        UF : 6, UT : 5,     CONFIG: 'N U T, 0, 0, 0',
       X = -330.7 mm, Y = 229.2 mm, Z = 498.2 mm,
       W = -5.3 deg, P = 20.5 deg,
    GP2:
        UF : 1, UT : 2,
       J1 = 0.0 deg, J2 = 0.0 deg
 };
P[405] {
    GP1:
        UF : 6, UT : 5,     CONFIG: 'N U T, 0, 0, 0',
 X = -313.7 mm, Y = 300.2 mm, Z = 498.2 mm,       W = -5.3 deg, P = 20.5 deg,
    GP2:
        UF : 1, UT : 2,
       J1 = 0.0 deg, J2 = 0.0 deg
 };
P[134] {
    GP1:
        UF : 6, UT : 5,     CONFIG: 'N U T, 0, 0, 0',
       X = -331.0 mm, Y = 230.3 mm, Z = 498.2 mm,
       W = -5.3 deg, P = 20.4 deg,
    GP2:
        UF : 1, UT : 2,
       J1 = 0.0 deg, J2 = 0.0 deg
 };
P[406] {
    GP1:
        UF : 6, UT : 5,     CONFIG: 'N U T, 0, 0, 0',
 X = -314.0 mm, Y = 301.3 mm, Z = 498.2 mm,       W = -5.3 deg, P = 20.4 deg,
    GP2:
        UF : 1, UT : 2,
       J1 = 0.0 deg, J2 = 0.0 deg
 };
P[135] {
    GP1:
        UF : 6, UT : 5,     CONFIG: 'N U T, 0, 0, 0',
       X = -333.4 mm, Y = 240.0 mm, Z = 498.2 mm,
       W = -5.7 deg, P = 19.9 deg,
    GP2:
        UF : 1, UT : 2,
       J1 = 0.0 deg, J2 = 0.0 deg
 };
P[407] {
    GP1:
        UF : 6, UT : 5,     CONFIG: 'N U T, 0, 0, 0',
 X = -316.4 mm, Y = 311.0 mm, Z = 498.2 mm,       W = -5.7 deg, P = 19.9 deg,
    GP2:
        UF : 1, UT : 2,
       J1 = 0.0 deg, J2 = 0.0 deg
 };
P[136] {
    GP1:
        UF : 6, UT : 5,     CONFIG: 'N U T, 0, 0, 0',
       X = -336.2 mm, Y = 249.6 mm, Z = 498.2 mm,
       W = -6.2 deg, P = 19.5 deg,
    GP2:
        UF : 1, UT : 2,
       J1 = 0.0 deg, J2 = 0.0 deg
 };
P[408] {
    GP1:
        UF : 6, UT : 5,     CONFIG: 'N U T, 0, 0, 0',
 X = -319.2 mm, Y = 320.6 mm, Z = 498.2 mm,       W = -6.2 deg, P = 19.5 deg,
    GP2:
        UF : 1, UT : 2,
       J1 = 0.0 deg, J2 = 0.0 deg
 };
P[137] {
    GP1:
        UF : 6, UT : 5,     CONFIG: 'N U T, 0, 0, 0',
       X = -339.1 mm, Y = 258.9 mm, Z = 498.2 mm,
       W = -6.7 deg, P = 19.1 deg,
    GP2:
        UF : 1, UT : 2,
       J1 = 0.0 deg, J2 = 0.0 deg
 };
P[409] {
    GP1:
        UF : 6, UT : 5,     CONFIG: 'N U T, 0, 0, 0',
 X = -322.1 mm, Y = 329.9 mm, Z = 498.2 mm,       W = -6.7 deg, P = 19.1 deg,
    GP2:
        UF : 1, UT : 2,
       J1 = 0.0 deg, J2 = 0.0 deg
 };
P[138] {
    GP1:
        UF : 6, UT : 5,     CONFIG: 'N U T, 0, 0, 0',
       X = -341.2 mm, Y = 265.0 mm, Z = 498.2 mm,
       W = -6.7 deg, P = 19.0 deg,
    GP2:
        UF : 1, UT : 2,
       J1 = 0.0 deg, J2 = 0.0 deg
 };
P[410] {
    GP1:
        UF : 6, UT : 5,     CONFIG: 'N U T, 0, 0, 0',
 X = -324.2 mm, Y = 336.0 mm, Z = 498.2 mm,       W = -6.7 deg, P = 19.0 deg,
    GP2:
        UF : 1, UT : 2,
       J1 = 0.0 deg, J2 = 0.0 deg
 };
P[139] {
    GP1:
        UF : 6, UT : 5,     CONFIG: 'N U T, 0, 0, 0',
       X = -341.9 mm, Y = 267.1 mm, Z = 498.2 mm,
       W = -7.2 deg, P = 18.7 deg,
    GP2:
        UF : 1, UT : 2,
       J1 = 0.0 deg, J2 = 0.0 deg
 };
P[411] {
    GP1:
        UF : 6, UT : 5,     CONFIG: 'N U T, 0, 0, 0',
 X = -324.9 mm, Y = 338.1 mm, Z = 498.2 mm,       W = -7.2 deg, P = 18.7 deg,
    GP2:
        UF : 1, UT : 2,
       J1 = 0.0 deg, J2 = 0.0 deg
 };
P[140] {
    GP1:
        UF : 6, UT : 5,     CONFIG: 'N U T, 0, 0, 0',
       X = -342.7 mm, Y = 269.1 mm, Z = 498.2 mm,
       W = -7.3 deg, P = 18.7 deg,
    GP2:
        UF : 1, UT : 2,
       J1 = 0.0 deg, J2 = 0.0 deg
 };
P[412] {
    GP1:
        UF : 6, UT : 5,     CONFIG: 'N U T, 0, 0, 0',
 X = -325.7 mm, Y = 340.1 mm, Z = 498.2 mm,       W = -7.3 deg, P = 18.7 deg,
    GP2:
        UF : 1, UT : 2,
       J1 = 0.0 deg, J2 = 0.0 deg
 };
P[141] {
    GP1:
        UF : 6, UT : 5,     CONFIG: 'N U T, 0, 0, 0',
       X = -344.3 mm, Y = 273.4 mm, Z = 498.2 mm,
       W = -7.2 deg, P = 18.6 deg,
    GP2:
        UF : 1, UT : 2,
       J1 = 0.0 deg, J2 = 0.0 deg
 };
P[413] {
    GP1:
        UF : 6, UT : 5,     CONFIG: 'N U T, 0, 0, 0',
 X = -327.3 mm, Y = 344.4 mm, Z = 498.2 mm,       W = -7.2 deg, P = 18.6 deg,
    GP2:
        UF : 1, UT : 2,
       J1 = 0.0 deg, J2 = 0.0 deg
 };
P[142] {
    GP1:
        UF : 6, UT : 5,     CONFIG: 'N U T, 0, 0, 0',
       X = -345.4 mm, Y = 276.1 mm, Z = 498.2 mm,
       W = -7.8 deg, P = 18.3 deg,
    GP2:
        UF : 1, UT : 2,
       J1 = 0.0 deg, J2 = 0.0 deg
 };
P[414] {
    GP1:
        UF : 6, UT : 5,     CONFIG: 'N U T, 0, 0, 0',
 X = -328.4 mm, Y = 347.1 mm, Z = 498.2 mm,       W = -7.8 deg, P = 18.3 deg,
    GP2:
        UF : 1, UT : 2,
       J1 = 0.0 deg, J2 = 0.0 deg
 };
P[143] {
    GP1:
        UF : 6, UT : 5,     CONFIG: 'N U T, 0, 0, 0',
       X = -346.5 mm, Y = 278.8 mm, Z = 498.2 mm,
       W = -7.9 deg, P = 18.2 deg,
    GP2:
        UF : 1, UT : 2,
       J1 = 0.0 deg, J2 = 0.0 deg
 };
P[415] {
    GP1:
        UF : 6, UT : 5,     CONFIG: 'N U T, 0, 0, 0',
 X = -329.5 mm, Y = 349.8 mm, Z = 498.2 mm,       W = -7.9 deg, P = 18.2 deg,
    GP2:
        UF : 1, UT : 2,
       J1 = 0.0 deg, J2 = 0.0 deg
 };
P[144] {
    GP1:
        UF : 6, UT : 5,     CONFIG: 'N U T, 0, 0, 0',
       X = -348.1 mm, Y = 282.6 mm, Z = 498.2 mm,
       W = -7.9 deg, P = 18.2 deg,
    GP2:
        UF : 1, UT : 2,
       J1 = 0.0 deg, J2 = 0.0 deg
 };
P[416] {
    GP1:
        UF : 6, UT : 5,     CONFIG: 'N U T, 0, 0, 0',
 X = -331.1 mm, Y = 353.6 mm, Z = 498.2 mm,       W = -7.9 deg, P = 18.2 deg,
    GP2:
        UF : 1, UT : 2,
       J1 = 0.0 deg, J2 = 0.0 deg
 };
P[145] {
    GP1:
        UF : 6, UT : 5,     CONFIG: 'N U T, 0, 0, 0',
       X = -349.4 mm, Y = 285.4 mm, Z = 498.2 mm,
       W = -8.5 deg, P = 17.9 deg,
    GP2:
        UF : 1, UT : 2,
       J1 = 0.0 deg, J2 = 0.0 deg
 };
P[417] {
    GP1:
        UF : 6, UT : 5,     CONFIG: 'N U T, 0, 0, 0',
 X = -332.4 mm, Y = 356.4 mm, Z = 498.2 mm,       W = -8.5 deg, P = 17.9 deg,
    GP2:
        UF : 1, UT : 2,
       J1 = 0.0 deg, J2 = 0.0 deg
 };
P[146] {
    GP1:
        UF : 6, UT : 5,     CONFIG: 'N U T, 0, 0, 0',
       X = -350.7 mm, Y = 288.2 mm, Z = 498.2 mm,
       W = -8.5 deg, P = 17.8 deg,
    GP2:
        UF : 1, UT : 2,
       J1 = 0.0 deg, J2 = 0.0 deg
 };
P[418] {
    GP1:
        UF : 6, UT : 5,     CONFIG: 'N U T, 0, 0, 0',
 X = -333.7 mm, Y = 359.2 mm, Z = 498.2 mm,       W = -8.5 deg, P = 17.8 deg,
    GP2:
        UF : 1, UT : 2,
       J1 = 0.0 deg, J2 = 0.0 deg
 };
P[147] {
    GP1:
        UF : 6, UT : 5,     CONFIG: 'N U T, 0, 0, 0',
       X = -352.3 mm, Y = 291.6 mm, Z = 498.2 mm,
       W = -8.4 deg, P = 17.7 deg,
    GP2:
        UF : 1, UT : 2,
       J1 = 0.0 deg, J2 = 0.0 deg
 };
P[419] {
    GP1:
        UF : 6, UT : 5,     CONFIG: 'N U T, 0, 0, 0',
 X = -335.3 mm, Y = 362.6 mm, Z = 498.2 mm,       W = -8.4 deg, P = 17.7 deg,
    GP2:
        UF : 1, UT : 2,
       J1 = 0.0 deg, J2 = 0.0 deg
 };
P[148] {
    GP1:
        UF : 6, UT : 5,     CONFIG: 'N U T, 0, 0, 0',
       X = -353.6 mm, Y = 294.5 mm, Z = 498.2 mm,
       W = -8.9 deg, P = 17.4 deg,
    GP2:
        UF : 1, UT : 2,
       J1 = 0.0 deg, J2 = 0.0 deg
 };
P[420] {
    GP1:
        UF : 6, UT : 5,     CONFIG: 'N U T, 0, 0, 0',
 X = -336.6 mm, Y = 365.5 mm, Z = 498.2 mm,       W = -8.9 deg, P = 17.4 deg,
    GP2:
        UF : 1, UT : 2,
       J1 = 0.0 deg, J2 = 0.0 deg
 };
P[149] {
    GP1:
        UF : 6, UT : 5,     CONFIG: 'N U T, 0, 0, 0',
       X = -355.0 mm, Y = 297.2 mm, Z = 498.2 mm,
       W = -9.0 deg, P = 17.3 deg,
    GP2:
        UF : 1, UT : 2,
       J1 = 0.0 deg, J2 = 0.0 deg
 };
P[421] {
    GP1:
        UF : 6, UT : 5,     CONFIG: 'N U T, 0, 0, 0',
 X = -338.0 mm, Y = 368.2 mm, Z = 498.2 mm,       W = -9.0 deg, P = 17.3 deg,
    GP2:
        UF : 1, UT : 2,
       J1 = 0.0 deg, J2 = 0.0 deg
 };
P[150] {
    GP1:
        UF : 6, UT : 5,     CONFIG: 'N U T, 0, 0, 0',
       X = -356.7 mm, Y = 300.5 mm, Z = 498.2 mm,
       W = -9.0 deg, P = 17.2 deg,
    GP2:
        UF : 1, UT : 2,
       J1 = 0.0 deg, J2 = 0.0 deg
 };
P[422] {
    GP1:
        UF : 6, UT : 5,     CONFIG: 'N U T, 0, 0, 0',
 X = -339.7 mm, Y = 371.5 mm, Z = 498.2 mm,       W = -9.0 deg, P = 17.2 deg,
    GP2:
        UF : 1, UT : 2,
       J1 = 0.0 deg, J2 = 0.0 deg
 };
P[151] {
    GP1:
        UF : 6, UT : 5,     CONFIG: 'N U T, 0, 0, 0',
       X = -358.2 mm, Y = 303.4 mm, Z = 498.2 mm,
       W = -9.4 deg, P = 16.9 deg,
    GP2:
        UF : 1, UT : 2,
       J1 = 0.0 deg, J2 = 0.0 deg
 };
P[423] {
    GP1:
        UF : 6, UT : 5,     CONFIG: 'N U T, 0, 0, 0',
 X = -341.2 mm, Y = 374.4 mm, Z = 498.2 mm,       W = -9.4 deg, P = 16.9 deg,
    GP2:
        UF : 1, UT : 2,
       J1 = 0.0 deg, J2 = 0.0 deg
 };
P[152] {
    GP1:
        UF : 6, UT : 5,     CONFIG: 'N U T, 0, 0, 0',
       X = -359.7 mm, Y = 306.2 mm, Z = 498.2 mm,
       W = -9.4 deg, P = 16.8 deg,
    GP2:
        UF : 1, UT : 2,
       J1 = 0.0 deg, J2 = 0.0 deg
 };
P[424] {
    GP1:
        UF : 6, UT : 5,     CONFIG: 'N U T, 0, 0, 0',
 X = -342.7 mm, Y = 377.2 mm, Z = 498.2 mm,       W = -9.4 deg, P = 16.8 deg,
    GP2:
        UF : 1, UT : 2,
       J1 = 0.0 deg, J2 = 0.0 deg
 };
P[153] {
    GP1:
        UF : 6, UT : 5,     CONFIG: 'N U T, 0, 0, 0',
       X = -361.4 mm, Y = 309.3 mm, Z = 498.2 mm,
       W = -9.4 deg, P = 16.7 deg,
    GP2:
        UF : 1, UT : 2,
       J1 = 0.0 deg, J2 = 0.0 deg
 };
P[425] {
    GP1:
        UF : 6, UT : 5,     CONFIG: 'N U T, 0, 0, 0',
 X = -344.4 mm, Y = 380.3 mm, Z = 498.2 mm,       W = -9.4 deg, P = 16.7 deg,
    GP2:
        UF : 1, UT : 2,
       J1 = 0.0 deg, J2 = 0.0 deg
 };
P[154] {
    GP1:
        UF : 6, UT : 5,     CONFIG: 'N U T, 0, 0, 0',
       X = -363.0 mm, Y = 312.1 mm, Z = 498.2 mm,
       W = -9.8 deg, P = 16.4 deg,
    GP2:
        UF : 1, UT : 2,
       J1 = 0.0 deg, J2 = 0.0 deg
 };
P[426] {
    GP1:
        UF : 6, UT : 5,     CONFIG: 'N U T, 0, 0, 0',
 X = -346.0 mm, Y = 383.1 mm, Z = 498.2 mm,       W = -9.8 deg, P = 16.4 deg,
    GP2:
        UF : 1, UT : 2,
       J1 = 0.0 deg, J2 = 0.0 deg
 };
P[155] {
    GP1:
        UF : 6, UT : 5,     CONFIG: 'N U T, 0, 0, 0',
       X = -368.0 mm, Y = 320.5 mm, Z = 498.2 mm,
       W = -10.0 deg, P = 15.8 deg,
    GP2:
        UF : 1, UT : 2,
       J1 = 0.0 deg, J2 = 0.0 deg
 };
P[427] {
    GP1:
        UF : 6, UT : 5,     CONFIG: 'N U T, 0, 0, 0',
 X = -351.0 mm, Y = 391.5 mm, Z = 498.2 mm,       W = -10.0 deg, P = 15.8 deg,
    GP2:
        UF : 1, UT : 2,
       J1 = 0.0 deg, J2 = 0.0 deg
 };
P[156] {
    GP1:
        UF : 6, UT : 5,     CONFIG: 'N U T, 0, 0, 0',
       X = -373.3 mm, Y = 328.8 mm, Z = 498.2 mm,
       W = -10.3 deg, P = 15.3 deg,
    GP2:
        UF : 1, UT : 2,
       J1 = 0.0 deg, J2 = 0.0 deg
 };
P[428] {
    GP1:
        UF : 6, UT : 5,     CONFIG: 'N U T, 0, 0, 0',
 X = -356.3 mm, Y = 399.8 mm, Z = 498.2 mm,       W = -10.3 deg, P = 15.3 deg,
    GP2:
        UF : 1, UT : 2,
       J1 = 0.0 deg, J2 = 0.0 deg
 };
P[157] {
    GP1:
        UF : 6, UT : 5,     CONFIG: 'N U T, 0, 0, 0',
       X = -378.8 mm, Y = 336.9 mm, Z = 498.2 mm,
       W = -10.5 deg, P = 14.7 deg,
    GP2:
        UF : 1, UT : 2,
       J1 = 0.0 deg, J2 = 0.0 deg
 };
P[429] {
    GP1:
        UF : 6, UT : 5,     CONFIG: 'N U T, 0, 0, 0',
 X = -361.8 mm, Y = 407.9 mm, Z = 498.2 mm,       W = -10.5 deg, P = 14.7 deg,
    GP2:
        UF : 1, UT : 2,
       J1 = 0.0 deg, J2 = 0.0 deg
 };
P[158] {
    GP1:
        UF : 6, UT : 5,     CONFIG: 'N U T, 0, 0, 0',
       X = -384.6 mm, Y = 344.9 mm, Z = 498.2 mm,
       W = -10.9 deg, P = 14.3 deg,
    GP2:
        UF : 1, UT : 2,
       J1 = 0.0 deg, J2 = 0.0 deg
 };
P[430] {
    GP1:
        UF : 6, UT : 5,     CONFIG: 'N U T, 0, 0, 0',
 X = -367.6 mm, Y = 415.9 mm, Z = 498.2 mm,       W = -10.9 deg, P = 14.3 deg,
    GP2:
        UF : 1, UT : 2,
       J1 = 0.0 deg, J2 = 0.0 deg
 };
P[159] {
    GP1:
        UF : 6, UT : 5,     CONFIG: 'N U T, 0, 0, 0',
       X = -390.6 mm, Y = 352.7 mm, Z = 498.2 mm,
       W = -11.0 deg, P = 13.7 deg,
    GP2:
        UF : 1, UT : 2,
       J1 = 0.0 deg, J2 = 0.0 deg
 };
P[431] {
    GP1:
        UF : 6, UT : 5,     CONFIG: 'N U T, 0, 0, 0',
 X = -373.6 mm, Y = 423.7 mm, Z = 498.2 mm,       W = -11.0 deg, P = 13.7 deg,
    GP2:
        UF : 1, UT : 2,
       J1 = 0.0 deg, J2 = 0.0 deg
 };
P[160] {
    GP1:
        UF : 6, UT : 5,     CONFIG: 'N U T, 0, 0, 0',
       X = -396.8 mm, Y = 360.3 mm, Z = 498.2 mm,
       W = -11.2 deg, P = 13.1 deg,
    GP2:
        UF : 1, UT : 2,
       J1 = 0.0 deg, J2 = 0.0 deg
 };
P[432] {
    GP1:
        UF : 6, UT : 5,     CONFIG: 'N U T, 0, 0, 0',
 X = -379.8 mm, Y = 431.3 mm, Z = 498.2 mm,       W = -11.2 deg, P = 13.1 deg,
    GP2:
        UF : 1, UT : 2,
       J1 = 0.0 deg, J2 = 0.0 deg
 };
P[161] {
    GP1:
        UF : 6, UT : 5,     CONFIG: 'N U T, 0, 0, 0',
       X = -403.2 mm, Y = 367.7 mm, Z = 498.2 mm,
       W = -11.4 deg, P = 12.7 deg,
    GP2:
        UF : 1, UT : 2,
       J1 = 0.0 deg, J2 = 0.0 deg
 };
P[433] {
    GP1:
        UF : 6, UT : 5,     CONFIG: 'N U T, 0, 0, 0',
 X = -386.2 mm, Y = 438.7 mm, Z = 498.2 mm,       W = -11.4 deg, P = 12.7 deg,
    GP2:
        UF : 1, UT : 2,
       J1 = 0.0 deg, J2 = 0.0 deg
 };
P[162] {
    GP1:
        UF : 6, UT : 5,     CONFIG: 'N U T, 0, 0, 0',
       X = -409.9 mm, Y = 374.9 mm, Z = 498.2 mm,
       W = -11.6 deg, P = 12.1 deg,
    GP2:
        UF : 1, UT : 2,
       J1 = 0.0 deg, J2 = 0.0 deg
 };
P[434] {
    GP1:
        UF : 6, UT : 5,     CONFIG: 'N U T, 0, 0, 0',
 X = -392.9 mm, Y = 445.9 mm, Z = 498.2 mm,       W = -11.6 deg, P = 12.1 deg,
    GP2:
        UF : 1, UT : 2,
       J1 = 0.0 deg, J2 = 0.0 deg
 };
P[163] {
    GP1:
        UF : 6, UT : 5,     CONFIG: 'N U T, 0, 0, 0',
       X = -416.7 mm, Y = 381.9 mm, Z = 498.2 mm,
       W = -11.5 deg, P = 11.5 deg,
    GP2:
        UF : 1, UT : 2,
       J1 = 0.0 deg, J2 = 0.0 deg
 };
P[435] {
    GP1:
        UF : 6, UT : 5,     CONFIG: 'N U T, 0, 0, 0',
 X = -399.7 mm, Y = 452.9 mm, Z = 498.2 mm,       W = -11.5 deg, P = 11.5 deg,
    GP2:
        UF : 1, UT : 2,
       J1 = 0.0 deg, J2 = 0.0 deg
 };
P[164] {
    GP1:
        UF : 6, UT : 5,     CONFIG: 'N U T, 0, 0, 0',
       X = -423.8 mm, Y = 388.7 mm, Z = 498.2 mm,
       W = -11.7 deg, P = 10.9 deg,
    GP2:
        UF : 1, UT : 2,
       J1 = 0.0 deg, J2 = 0.0 deg
 };
P[436] {
    GP1:
        UF : 6, UT : 5,     CONFIG: 'N U T, 0, 0, 0',
 X = -406.8 mm, Y = 459.7 mm, Z = 498.2 mm,       W = -11.7 deg, P = 10.9 deg,
    GP2:
        UF : 1, UT : 2,
       J1 = 0.0 deg, J2 = 0.0 deg
 };
P[165] {
    GP1:
        UF : 6, UT : 5,     CONFIG: 'N U T, 0, 0, 0',
       X = -431.1 mm, Y = 395.2 mm, Z = 498.2 mm,
       W = -11.7 deg, P = 10.3 deg,
    GP2:
        UF : 1, UT : 2,
       J1 = 0.0 deg, J2 = 0.0 deg
 };
P[437] {
    GP1:
        UF : 6, UT : 5,     CONFIG: 'N U T, 0, 0, 0',
 X = -414.1 mm, Y = 466.2 mm, Z = 498.2 mm,       W = -11.7 deg, P = 10.3 deg,
    GP2:
        UF : 1, UT : 2,
       J1 = 0.0 deg, J2 = 0.0 deg
 };
P[166] {
    GP1:
        UF : 6, UT : 5,     CONFIG: 'N U T, 0, 0, 0',
       X = -434.4 mm, Y = 398.1 mm, Z = 498.2 mm,
       W = -11.7 deg, P = 10.1 deg,
    GP2:
        UF : 1, UT : 2,
       J1 = 0.0 deg, J2 = 0.0 deg
 };
P[438] {
    GP1:
        UF : 6, UT : 5,     CONFIG: 'N U T, 0, 0, 0',
 X = -417.4 mm, Y = 469.1 mm, Z = 498.2 mm,       W = -11.7 deg, P = 10.1 deg,
    GP2:
        UF : 1, UT : 2,
       J1 = 0.0 deg, J2 = 0.0 deg
 };
P[167] {
    GP1:
        UF : 6, UT : 5,     CONFIG: 'N U T, 0, 0, 0',
       X = -436.8 mm, Y = 400.2 mm, Z = 498.2 mm,
       W = -11.8 deg, P = 10.1 deg,
    GP2:
        UF : 1, UT : 2,
       J1 = 0.0 deg, J2 = 0.0 deg
 };
P[439] {
    GP1:
        UF : 6, UT : 5,     CONFIG: 'N U T, 0, 0, 0',
 X = -419.8 mm, Y = 471.2 mm, Z = 498.2 mm,       W = -11.8 deg, P = 10.1 deg,
    GP2:
        UF : 1, UT : 2,
       J1 = 0.0 deg, J2 = 0.0 deg
 };
P[168] {
    GP1:
        UF : 6, UT : 5,     CONFIG: 'N U T, 0, 0, 0',
       X = -438.2 mm, Y = 401.3 mm, Z = 498.2 mm,
       W = -11.5 deg, P = 10.7 deg,
    GP2:
        UF : 1, UT : 2,
       J1 = 0.0 deg, J2 = 0.0 deg
 };
P[440] {
    GP1:
        UF : 6, UT : 5,     CONFIG: 'N U T, 0, 0, 0',
 X = -421.2 mm, Y = 472.3 mm, Z = 498.2 mm,       W = -11.5 deg, P = 10.7 deg,
    GP2:
        UF : 1, UT : 2,
       J1 = 0.0 deg, J2 = 0.0 deg
 };
P[169] {
    GP1:
        UF : 6, UT : 5,     CONFIG: 'N U T, 0, 0, 0',
       X = -439.0 mm, Y = 402.1 mm, Z = 498.2 mm,
       W = -11.1 deg, P = 11.0 deg,
    GP2:
        UF : 1, UT : 2,
       J1 = 0.0 deg, J2 = 0.0 deg
 };
P[441] {
    GP1:
        UF : 6, UT : 5,     CONFIG: 'N U T, 0, 0, 0',
 X = -422.0 mm, Y = 473.1 mm, Z = 498.2 mm,       W = -11.1 deg, P = 11.0 deg,
    GP2:
        UF : 1, UT : 2,
       J1 = 0.0 deg, J2 = 0.0 deg
 };
P[170] {
    GP1:
        UF : 6, UT : 5,     CONFIG: 'N U T, 0, 0, 0',
       X = -439.8 mm, Y = 402.9 mm, Z = 498.2 mm,
       W = -10.4 deg, P = 11.8 deg,
    GP2:
        UF : 1, UT : 2,
       J1 = 0.0 deg, J2 = 0.0 deg
 };
P[442] {
    GP1:
        UF : 6, UT : 5,     CONFIG: 'N U T, 0, 0, 0',
 X = -422.8 mm, Y = 473.9 mm, Z = 498.2 mm,       W = -10.4 deg, P = 11.8 deg,
    GP2:
        UF : 1, UT : 2,
       J1 = 0.0 deg, J2 = 0.0 deg
 };
P[171] {
    GP1:
        UF : 6, UT : 5,     CONFIG: 'N U T, 0, 0, 0',
       X = -440.4 mm, Y = 403.8 mm, Z = 498.2 mm,
       W = -9.8 deg, P = 12.5 deg,
    GP2:
        UF : 1, UT : 2,
       J1 = 0.0 deg, J2 = 0.0 deg
 };
P[443] {
    GP1:
        UF : 6, UT : 5,     CONFIG: 'N U T, 0, 0, 0',
 X = -423.4 mm, Y = 474.8 mm, Z = 498.2 mm,       W = -9.8 deg, P = 12.5 deg,
    GP2:
        UF : 1, UT : 2,
       J1 = 0.0 deg, J2 = 0.0 deg
 };
P[172] {
    GP1:
        UF : 6, UT : 5,     CONFIG: 'N U T, 0, 0, 0',
       X = -440.7 mm, Y = 404.2 mm, Z = 498.2 mm,
       W = -9.6 deg, P = 12.8 deg,
    GP2:
        UF : 1, UT : 2,
       J1 = 0.0 deg, J2 = 0.0 deg
 };
P[444] {
    GP1:
        UF : 6, UT : 5,     CONFIG: 'N U T, 0, 0, 0',
 X = -423.7 mm, Y = 475.2 mm, Z = 498.2 mm,       W = -9.6 deg, P = 12.8 deg,
    GP2:
        UF : 1, UT : 2,
       J1 = 0.0 deg, J2 = 0.0 deg
 };
P[173] {
    GP1:
        UF : 6, UT : 5,     CONFIG: 'N U T, 0, 0, 0',
       X = -441.0 mm, Y = 404.6 mm, Z = 498.2 mm,
       W = -9.3 deg, P = 12.9 deg,
    GP2:
        UF : 1, UT : 2,
       J1 = 0.0 deg, J2 = 0.0 deg
 };
P[445] {
    GP1:
        UF : 6, UT : 5,     CONFIG: 'N U T, 0, 0, 0',
 X = -424.0 mm, Y = 475.6 mm, Z = 498.2 mm,       W = -9.3 deg, P = 12.9 deg,
    GP2:
        UF : 1, UT : 2,
       J1 = 0.0 deg, J2 = 0.0 deg
 };
P[174] {
    GP1:
        UF : 6, UT : 5,     CONFIG: 'N U T, 0, 0, 0',
       X = -441.3 mm, Y = 404.9 mm, Z = 498.2 mm,
       W = -9.1 deg, P = 13.1 deg,
    GP2:
        UF : 1, UT : 2,
       J1 = 0.0 deg, J2 = 0.0 deg
 };
P[446] {
    GP1:
        UF : 6, UT : 5,     CONFIG: 'N U T, 0, 0, 0',
 X = -424.3 mm, Y = 475.9 mm, Z = 498.2 mm,       W = -9.1 deg, P = 13.1 deg,
    GP2:
        UF : 1, UT : 2,
       J1 = 0.0 deg, J2 = 0.0 deg
 };
P[175] {
    GP1:
        UF : 6, UT : 5,     CONFIG: 'N U T, 0, 0, 0',
       X = -441.6 mm, Y = 405.3 mm, Z = 498.2 mm,
       W = -8.9 deg, P = 13.3 deg,
    GP2:
        UF : 1, UT : 2,
       J1 = 0.0 deg, J2 = 0.0 deg
 };
P[447] {
    GP1:
        UF : 6, UT : 5,     CONFIG: 'N U T, 0, 0, 0',
 X = -424.6 mm, Y = 476.3 mm, Z = 498.2 mm,       W = -8.9 deg, P = 13.3 deg,
    GP2:
        UF : 1, UT : 2,
       J1 = 0.0 deg, J2 = 0.0 deg
 };
P[176] {
    GP1:
        UF : 6, UT : 5,     CONFIG: 'N U T, 0, 0, 0',
       X = -441.7 mm, Y = 405.5 mm, Z = 498.2 mm,
       W = -8.6 deg, P = 13.5 deg,
    GP2:
        UF : 1, UT : 2,
       J1 = 0.0 deg, J2 = 0.0 deg
 };
P[448] {
    GP1:
        UF : 6, UT : 5,     CONFIG: 'N U T, 0, 0, 0',
 X = -424.7 mm, Y = 476.5 mm, Z = 498.2 mm,       W = -8.6 deg, P = 13.5 deg,
    GP2:
        UF : 1, UT : 2,
       J1 = 0.0 deg, J2 = 0.0 deg
 };
P[177] {
    GP1:
        UF : 6, UT : 5,     CONFIG: 'N U T, 0, 0, 0',
       X = -441.8 mm, Y = 405.8 mm, Z = 498.2 mm,
       W = -8.3 deg, P = 13.6 deg,
    GP2:
        UF : 1, UT : 2,
       J1 = 0.0 deg, J2 = 0.0 deg
 };
P[449] {
    GP1:
        UF : 6, UT : 5,     CONFIG: 'N U T, 0, 0, 0',
 X = -424.8 mm, Y = 476.8 mm, Z = 498.2 mm,       W = -8.3 deg, P = 13.6 deg,
    GP2:
        UF : 1, UT : 2,
       J1 = 0.0 deg, J2 = 0.0 deg
 };
P[178] {
    GP1:
        UF : 6, UT : 5,     CONFIG: 'N U T, 0, 0, 0',
       X = -442.0 mm, Y = 406.0 mm, Z = 498.2 mm,
       W = -8.0 deg, P = 13.8 deg,
    GP2:
        UF : 1, UT : 2,
       J1 = 0.0 deg, J2 = 0.0 deg
 };
P[450] {
    GP1:
        UF : 6, UT : 5,     CONFIG: 'N U T, 0, 0, 0',
 X = -425.0 mm, Y = 477.0 mm, Z = 498.2 mm,       W = -8.0 deg, P = 13.8 deg,
    GP2:
        UF : 1, UT : 2,
       J1 = 0.0 deg, J2 = 0.0 deg
 };
P[179] {
    GP1:
        UF : 6, UT : 5,     CONFIG: 'N U T, 0, 0, 0',
       X = -442.1 mm, Y = 406.2 mm, Z = 498.2 mm,
       W = -7.7 deg, P = 14.0 deg,
    GP2:
        UF : 1, UT : 2,
       J1 = 0.0 deg, J2 = 0.0 deg
 };
P[451] {
    GP1:
        UF : 6, UT : 5,     CONFIG: 'N U T, 0, 0, 0',
 X = -425.1 mm, Y = 477.2 mm, Z = 498.2 mm,       W = -7.7 deg, P = 14.0 deg,
    GP2:
        UF : 1, UT : 2,
       J1 = 0.0 deg, J2 = 0.0 deg
 };
P[180] {
    GP1:
        UF : 6, UT : 5,     CONFIG: 'N U T, 0, 0, 0',
       X = -442.5 mm, Y = 407.1 mm, Z = 498.2 mm,
       W = -7.2 deg, P = 14.1 deg,
    GP2:
        UF : 1, UT : 2,
       J1 = 0.0 deg, J2 = 0.0 deg
 };
P[452] {
    GP1:
        UF : 6, UT : 5,     CONFIG: 'N U T, 0, 0, 0',
 X = -425.5 mm, Y = 478.1 mm, Z = 498.2 mm,       W = -7.2 deg, P = 14.1 deg,
    GP2:
        UF : 1, UT : 2,
       J1 = 0.0 deg, J2 = 0.0 deg
 };
P[181] {
    GP1:
        UF : 6, UT : 5,     CONFIG: 'N U T, 0, 0, 0',
       X = -442.9 mm, Y = 407.8 mm, Z = 498.2 mm,
       W = -6.9 deg, P = 14.2 deg,
    GP2:
        UF : 1, UT : 2,
       J1 = 0.0 deg, J2 = 0.0 deg
 };
P[453] {
    GP1:
        UF : 6, UT : 5,     CONFIG: 'N U T, 0, 0, 0',
 X = -425.9 mm, Y = 478.8 mm, Z = 498.2 mm,       W = -6.9 deg, P = 14.2 deg,
    GP2:
        UF : 1, UT : 2,
       J1 = 0.0 deg, J2 = 0.0 deg
 };
P[182] {
    GP1:
        UF : 6, UT : 5,     CONFIG: 'N U T, 0, 0, 0',
       X = -443.2 mm, Y = 408.4 mm, Z = 498.2 mm,
       W = -6.0 deg, P = 14.6 deg,
    GP2:
        UF : 1, UT : 2,
       J1 = 0.0 deg, J2 = 0.0 deg
 };
P[454] {
    GP1:
        UF : 6, UT : 5,     CONFIG: 'N U T, 0, 0, 0',
 X = -426.2 mm, Y = 479.4 mm, Z = 498.2 mm,       W = -6.0 deg, P = 14.6 deg,
    GP2:
        UF : 1, UT : 2,
       J1 = 0.0 deg, J2 = 0.0 deg
 };
P[183] {
    GP1:
        UF : 6, UT : 5,     CONFIG: 'N U T, 0, 0, 0',
       X = -443.3 mm, Y = 408.9 mm, Z = 498.2 mm,
       W = -5.2 deg, P = 14.7 deg,
    GP2:
        UF : 1, UT : 2,
       J1 = 0.0 deg, J2 = 0.0 deg
 };
P[455] {
    GP1:
        UF : 6, UT : 5,     CONFIG: 'N U T, 0, 0, 0',
 X = -426.3 mm, Y = 479.9 mm, Z = 498.2 mm,       W = -5.2 deg, P = 14.7 deg,
    GP2:
        UF : 1, UT : 2,
       J1 = 0.0 deg, J2 = 0.0 deg
 };
P[184] {
    GP1:
        UF : 6, UT : 5,     CONFIG: 'N U T, 0, 0, 0',
       X = -443.7 mm, Y = 410.1 mm, Z = 498.2 mm,
       W = -4.4 deg, P = 14.6 deg,
    GP2:
        UF : 1, UT : 2,
       J1 = 0.0 deg, J2 = 0.0 deg
 };
P[456] {
    GP1:
        UF : 6, UT : 5,     CONFIG: 'N U T, 0, 0, 0',
 X = -426.7 mm, Y = 481.1 mm, Z = 498.2 mm,       W = -4.4 deg, P = 14.6 deg,
    GP2:
        UF : 1, UT : 2,
       J1 = 0.0 deg, J2 = 0.0 deg
 };
P[185] {
    GP1:
        UF : 6, UT : 5,     CONFIG: 'N U T, 0, 0, 0',
       X = -444.0 mm, Y = 411.0 mm, Z = 498.2 mm,
       W = -3.9 deg, P = 14.7 deg,
    GP2:
        UF : 1, UT : 2,
       J1 = 0.0 deg, J2 = 0.0 deg
 };
P[457] {
    GP1:
        UF : 6, UT : 5,     CONFIG: 'N U T, 0, 0, 0',
 X = -427.0 mm, Y = 482.0 mm, Z = 498.2 mm,       W = -3.9 deg, P = 14.7 deg,
    GP2:
        UF : 1, UT : 2,
       J1 = 0.0 deg, J2 = 0.0 deg
 };
P[186] {
    GP1:
        UF : 6, UT : 5,     CONFIG: 'N U T, 0, 0, 0',
       X = -444.0 mm, Y = 411.2 mm, Z = 498.2 mm,
       W = -3.6 deg, P = 14.6 deg,
    GP2:
        UF : 1, UT : 2,
       J1 = 0.0 deg, J2 = 0.0 deg
 };
P[458] {
    GP1:
        UF : 6, UT : 5,     CONFIG: 'N U T, 0, 0, 0',
 X = -427.0 mm, Y = 482.2 mm, Z = 498.2 mm,       W = -3.6 deg, P = 14.6 deg,
    GP2:
        UF : 1, UT : 2,
       J1 = 0.0 deg, J2 = 0.0 deg
 };
P[187] {
    GP1:
        UF : 6, UT : 5,     CONFIG: 'N U T, 0, 0, 0',
       X = -444.1 mm, Y = 411.4 mm, Z = 498.2 mm,
       W = -3.2 deg, P = 14.6 deg,
    GP2:
        UF : 1, UT : 2,
       J1 = 0.0 deg, J2 = 0.0 deg
 };
P[459] {
    GP1:
        UF : 6, UT : 5,     CONFIG: 'N U T, 0, 0, 0',
 X = -427.1 mm, Y = 482.4 mm, Z = 498.2 mm,       W = -3.2 deg, P = 14.6 deg,
    GP2:
        UF : 1, UT : 2,
       J1 = 0.0 deg, J2 = 0.0 deg
 };
P[188] {
    GP1:
        UF : 6, UT : 5,     CONFIG: 'N U T, 0, 0, 0',
       X = -444.1 mm, Y = 411.6 mm, Z = 498.2 mm,
       W = -2.8 deg, P = 14.6 deg,
    GP2:
        UF : 1, UT : 2,
       J1 = 0.0 deg, J2 = 0.0 deg
 };
P[460] {
    GP1:
        UF : 6, UT : 5,     CONFIG: 'N U T, 0, 0, 0',
 X = -427.1 mm, Y = 482.6 mm, Z = 498.2 mm,       W = -2.8 deg, P = 14.6 deg,
    GP2:
        UF : 1, UT : 2,
       J1 = 0.0 deg, J2 = 0.0 deg
 };
P[189] {
    GP1:
        UF : 6, UT : 5,     CONFIG: 'N U T, 0, 0, 0',
       X = -444.2 mm, Y = 411.8 mm, Z = 498.2 mm,
       W = -2.5 deg, P = 14.6 deg,
    GP2:
        UF : 1, UT : 2,
       J1 = 0.0 deg, J2 = 0.0 deg
 };
P[461] {
    GP1:
        UF : 6, UT : 5,     CONFIG: 'N U T, 0, 0, 0',
 X = -427.2 mm, Y = 482.8 mm, Z = 498.2 mm,       W = -2.5 deg, P = 14.6 deg,
    GP2:
        UF : 1, UT : 2,
       J1 = 0.0 deg, J2 = 0.0 deg
 };
P[190] {
    GP1:
        UF : 6, UT : 5,     CONFIG: 'N U T, 0, 0, 0',
       X = -444.3 mm, Y = 412.7 mm, Z = 498.2 mm,
       W = -2.0 deg, P = 14.2 deg,
    GP2:
        UF : 1, UT : 2,
       J1 = 0.0 deg, J2 = 0.0 deg
 };
P[462] {
    GP1:
        UF : 6, UT : 5,     CONFIG: 'N U T, 0, 0, 0',
 X = -427.3 mm, Y = 483.7 mm, Z = 498.2 mm,       W = -2.0 deg, P = 14.2 deg,
    GP2:
        UF : 1, UT : 2,
       J1 = 0.0 deg, J2 = 0.0 deg
 };
P[191] {
    GP1:
        UF : 6, UT : 5,     CONFIG: 'N U T, 0, 0, 0',
       X = -444.4 mm, Y = 414.0 mm, Z = 498.2 mm,
       W = -0.9 deg, P = 13.9 deg,
    GP2:
        UF : 1, UT : 2,
       J1 = 0.0 deg, J2 = 0.0 deg
 };
P[463] {
    GP1:
        UF : 6, UT : 5,     CONFIG: 'N U T, 0, 0, 0',
 X = -427.4 mm, Y = 485.0 mm, Z = 498.2 mm,       W = -0.9 deg, P = 13.9 deg,
    GP2:
        UF : 1, UT : 2,
       J1 = 0.0 deg, J2 = 0.0 deg
 };
P[192] {
    GP1:
        UF : 6, UT : 5,     CONFIG: 'N U T, 0, 0, 0',
       X = -444.4 mm, Y = 414.3 mm, Z = 498.2 mm,
       W = -0.6 deg, P = 13.7 deg,
    GP2:
        UF : 1, UT : 2,
       J1 = 0.0 deg, J2 = 0.0 deg
 };
P[464] {
    GP1:
        UF : 6, UT : 5,     CONFIG: 'N U T, 0, 0, 0',
 X = -427.4 mm, Y = 485.3 mm, Z = 498.2 mm,       W = -0.6 deg, P = 13.7 deg,
    GP2:
        UF : 1, UT : 2,
       J1 = 0.0 deg, J2 = 0.0 deg
 };
P[193] {
    GP1:
        UF : 6, UT : 5,     CONFIG: 'N U T, 0, 0, 0',
       X = -444.4 mm, Y = 414.6 mm, Z = 498.2 mm,
       W = -0.4 deg, P = 13.5 deg,
    GP2:
        UF : 1, UT : 2,
       J1 = 0.0 deg, J2 = 0.0 deg
 };
P[465] {
    GP1:
        UF : 6, UT : 5,     CONFIG: 'N U T, 0, 0, 0',
 X = -427.4 mm, Y = 485.6 mm, Z = 498.2 mm,       W = -0.4 deg, P = 13.5 deg,
    GP2:
        UF : 1, UT : 2,
       J1 = 0.0 deg, J2 = 0.0 deg
 };
P[194] {
    GP1:
        UF : 6, UT : 5,     CONFIG: 'N U T, 0, 0, 0',
       X = -444.5 mm, Y = 414.9 mm, Z = 498.2 mm,
       W = -0.1 deg, P = 13.4 deg,
    GP2:
        UF : 1, UT : 2,
       J1 = 0.0 deg, J2 = 0.0 deg
 };
P[466] {
    GP1:
        UF : 6, UT : 5,     CONFIG: 'N U T, 0, 0, 0',
 X = -427.5 mm, Y = 485.9 mm, Z = 498.2 mm,       W = -0.1 deg, P = 13.4 deg,
    GP2:
        UF : 1, UT : 2,
       J1 = 0.0 deg, J2 = 0.0 deg
 };
P[195] {
    GP1:
        UF : 6, UT : 5,     CONFIG: 'N U T, 0, 0, 0',
       X = -444.5 mm, Y = 415.3 mm, Z = 498.2 mm,
       W = 0.1 deg, P = 13.2 deg,
    GP2:
        UF : 1, UT : 2,
       J1 = 0.0 deg, J2 = 0.0 deg
 };
P[467] {
    GP1:
        UF : 6, UT : 5,     CONFIG: 'N U T, 0, 0, 0',
 X = -427.5 mm, Y = 486.3 mm, Z = 498.2 mm,       W = 0.1 deg, P = 13.2 deg,
    GP2:
        UF : 1, UT : 2,
       J1 = 0.0 deg, J2 = 0.0 deg
 };
P[196] {
    GP1:
        UF : 6, UT : 5,     CONFIG: 'N U T, 0, 0, 0',
       X = -444.4 mm, Y = 416.3 mm, Z = 498.2 mm,
       W = 0.6 deg, P = 12.9 deg,
    GP2:
        UF : 1, UT : 2,
       J1 = 0.0 deg, J2 = 0.0 deg
 };
P[468] {
    GP1:
        UF : 6, UT : 5,     CONFIG: 'N U T, 0, 0, 0',
 X = -427.4 mm, Y = 487.3 mm, Z = 498.2 mm,       W = 0.6 deg, P = 12.9 deg,
    GP2:
        UF : 1, UT : 2,
       J1 = 0.0 deg, J2 = 0.0 deg
 };
P[197] {
    GP1:
        UF : 6, UT : 5,     CONFIG: 'N U T, 0, 0, 0',
       X = -444.4 mm, Y = 416.6 mm, Z = 498.2 mm,
       W = 0.9 deg, P = 12.7 deg,
    GP2:
        UF : 1, UT : 2,
       J1 = 0.0 deg, J2 = 0.0 deg
 };
P[469] {
    GP1:
        UF : 6, UT : 5,     CONFIG: 'N U T, 0, 0, 0',
 X = -427.4 mm, Y = 487.6 mm, Z = 498.2 mm,       W = 0.9 deg, P = 12.7 deg,
    GP2:
        UF : 1, UT : 2,
       J1 = 0.0 deg, J2 = 0.0 deg
 };
P[198] {
    GP1:
        UF : 6, UT : 5,     CONFIG: 'N U T, 0, 0, 0',
       X = -444.4 mm, Y = 416.9 mm, Z = 498.2 mm,
       W = 1.2 deg, P = 12.5 deg,
    GP2:
        UF : 1, UT : 2,
       J1 = 0.0 deg, J2 = 0.0 deg
 };
P[470] {
    GP1:
        UF : 6, UT : 5,     CONFIG: 'N U T, 0, 0, 0',
 X = -427.4 mm, Y = 487.9 mm, Z = 498.2 mm,       W = 1.2 deg, P = 12.5 deg,
    GP2:
        UF : 1, UT : 2,
       J1 = 0.0 deg, J2 = 0.0 deg
 };
P[199] {
    GP1:
        UF : 6, UT : 5,     CONFIG: 'N U T, 0, 0, 0',
       X = -444.4 mm, Y = 417.2 mm, Z = 498.2 mm,
       W = 1.5 deg, P = 12.4 deg,
    GP2:
        UF : 1, UT : 2,
       J1 = 0.0 deg, J2 = 0.0 deg
 };
P[471] {
    GP1:
        UF : 6, UT : 5,     CONFIG: 'N U T, 0, 0, 0',
 X = -427.4 mm, Y = 488.2 mm, Z = 498.2 mm,       W = 1.5 deg, P = 12.4 deg,
    GP2:
        UF : 1, UT : 2,
       J1 = 0.0 deg, J2 = 0.0 deg
 };
P[200] {
    GP1:
        UF : 6, UT : 5,     CONFIG: 'N U T, 0, 0, 0',
       X = -444.3 mm, Y = 417.5 mm, Z = 498.2 mm,
       W = 1.8 deg, P = 12.2 deg,
    GP2:
        UF : 1, UT : 2,
       J1 = 0.0 deg, J2 = 0.0 deg
 };
P[472] {
    GP1:
        UF : 6, UT : 5,     CONFIG: 'N U T, 0, 0, 0',
 X = -427.3 mm, Y = 488.5 mm, Z = 498.2 mm,       W = 1.8 deg, P = 12.2 deg,
    GP2:
        UF : 1, UT : 2,
       J1 = 0.0 deg, J2 = 0.0 deg
 };
P[201] {
    GP1:
        UF : 6, UT : 5,     CONFIG: 'N U T, 0, 0, 0',
       X = -444.1 mm, Y = 418.6 mm, Z = 498.2 mm,
       W = 2.2 deg, P = 11.0 deg,
    GP2:
        UF : 1, UT : 2,
       J1 = 0.0 deg, J2 = 0.0 deg
 };
P[473] {
    GP1:
        UF : 6, UT : 5,     CONFIG: 'N U T, 0, 0, 0',
 X = -427.1 mm, Y = 489.6 mm, Z = 498.2 mm,       W = 2.2 deg, P = 11.0 deg,
    GP2:
        UF : 1, UT : 2,
       J1 = 0.0 deg, J2 = 0.0 deg
 };
P[202] {
    GP1:
        UF : 6, UT : 5,     CONFIG: 'N U T, 0, 0, 0',
       X = -443.9 mm, Y = 419.8 mm, Z = 498.2 mm,
       W = 2.5 deg, P = 10.2 deg,
    GP2:
        UF : 1, UT : 2,
       J1 = 0.0 deg, J2 = 0.0 deg
 };
P[474] {
    GP1:
        UF : 6, UT : 5,     CONFIG: 'N U T, 0, 0, 0',
 X = -426.9 mm, Y = 490.8 mm, Z = 498.2 mm,       W = 2.5 deg, P = 10.2 deg,
    GP2:
        UF : 1, UT : 2,
       J1 = 0.0 deg, J2 = 0.0 deg
 };
P[203] {
    GP1:
        UF : 6, UT : 5,     CONFIG: 'N U T, 0, 0, 0',
       X = -443.8 mm, Y = 420.0 mm, Z = 498.2 mm,
       W = 2.7 deg, P = 10.0 deg,
    GP2:
        UF : 1, UT : 2,
       J1 = 0.0 deg, J2 = 0.0 deg
 };
P[475] {
    GP1:
        UF : 6, UT : 5,     CONFIG: 'N U T, 0, 0, 0',
 X = -426.8 mm, Y = 491.0 mm, Z = 498.2 mm,       W = 2.7 deg, P = 10.0 deg,
    GP2:
        UF : 1, UT : 2,
       J1 = 0.0 deg, J2 = 0.0 deg
 };
P[204] {
    GP1:
        UF : 6, UT : 5,     CONFIG: 'N U T, 0, 0, 0',
       X = -443.8 mm, Y = 420.2 mm, Z = 498.2 mm,
       W = 2.9 deg, P = 9.9 deg,
    GP2:
        UF : 1, UT : 2,
       J1 = 0.0 deg, J2 = 0.0 deg
 };
P[476] {
    GP1:
        UF : 6, UT : 5,     CONFIG: 'N U T, 0, 0, 0',
 X = -426.8 mm, Y = 491.2 mm, Z = 498.2 mm,       W = 2.9 deg, P = 9.9 deg,
    GP2:
        UF : 1, UT : 2,
       J1 = 0.0 deg, J2 = 0.0 deg
 };
P[205] {
    GP1:
        UF : 6, UT : 5,     CONFIG: 'N U T, 0, 0, 0',
       X = -443.7 mm, Y = 420.4 mm, Z = 498.2 mm,
       W = 3.0 deg, P = 9.7 deg,
    GP2:
        UF : 1, UT : 2,
       J1 = 0.0 deg, J2 = 0.0 deg
 };
P[477] {
    GP1:
        UF : 6, UT : 5,     CONFIG: 'N U T, 0, 0, 0',
 X = -426.7 mm, Y = 491.4 mm, Z = 498.2 mm,       W = 3.0 deg, P = 9.7 deg,
    GP2:
        UF : 1, UT : 2,
       J1 = 0.0 deg, J2 = 0.0 deg
 };
P[206] {
    GP1:
        UF : 6, UT : 5,     CONFIG: 'N U T, 0, 0, 0',
       X = -443.6 mm, Y = 420.7 mm, Z = 498.2 mm,
       W = 3.2 deg, P = 9.5 deg,
    GP2:
        UF : 1, UT : 2,
       J1 = 0.0 deg, J2 = 0.0 deg
 };
P[478] {
    GP1:
        UF : 6, UT : 5,     CONFIG: 'N U T, 0, 0, 0',
 X = -426.6 mm, Y = 491.7 mm, Z = 498.2 mm,       W = 3.2 deg, P = 9.5 deg,
    GP2:
        UF : 1, UT : 2,
       J1 = 0.0 deg, J2 = 0.0 deg
 };
P[207] {
    GP1:
        UF : 6, UT : 5,     CONFIG: 'N U T, 0, 0, 0',
       X = -443.3 mm, Y = 421.5 mm, Z = 498.2 mm,
       W = 3.4 deg, P = 8.9 deg,
    GP2:
        UF : 1, UT : 2,
       J1 = 0.0 deg, J2 = 0.0 deg
 };
P[479] {
    GP1:
        UF : 6, UT : 5,     CONFIG: 'N U T, 0, 0, 0',
 X = -426.3 mm, Y = 492.5 mm, Z = 498.2 mm,       W = 3.4 deg, P = 8.9 deg,
    GP2:
        UF : 1, UT : 2,
       J1 = 0.0 deg, J2 = 0.0 deg
 };
P[208] {
    GP1:
        UF : 6, UT : 5,     CONFIG: 'N U T, 0, 0, 0',
       X = -442.8 mm, Y = 422.8 mm, Z = 498.2 mm,
       W = 3.5 deg, P = 7.9 deg,
    GP2:
        UF : 1, UT : 2,
       J1 = 0.0 deg, J2 = 0.0 deg
 };
P[480] {
    GP1:
        UF : 6, UT : 5,     CONFIG: 'N U T, 0, 0, 0',
 X = -425.8 mm, Y = 493.8 mm, Z = 498.2 mm,       W = 3.5 deg, P = 7.9 deg,
    GP2:
        UF : 1, UT : 2,
       J1 = 0.0 deg, J2 = 0.0 deg
 };
P[209] {
    GP1:
        UF : 6, UT : 5,     CONFIG: 'N U T, 0, 0, 0',
       X = -442.7 mm, Y = 423.0 mm, Z = 498.2 mm,
       W = 3.5 deg, P = 7.7 deg,
    GP2:
        UF : 1, UT : 2,
       J1 = 0.0 deg, J2 = 0.0 deg
 };
P[481] {
    GP1:
        UF : 6, UT : 5,     CONFIG: 'N U T, 0, 0, 0',
 X = -425.7 mm, Y = 494.0 mm, Z = 498.2 mm,       W = 3.5 deg, P = 7.7 deg,
    GP2:
        UF : 1, UT : 2,
       J1 = 0.0 deg, J2 = 0.0 deg
 };
P[210] {
    GP1:
        UF : 6, UT : 5,     CONFIG: 'N U T, 0, 0, 0',
       X = -442.6 mm, Y = 423.3 mm, Z = 498.2 mm,
       W = 3.6 deg, P = 7.4 deg,
    GP2:
        UF : 1, UT : 2,
       J1 = 0.0 deg, J2 = 0.0 deg
 };
P[482] {
    GP1:
        UF : 6, UT : 5,     CONFIG: 'N U T, 0, 0, 0',
 X = -425.6 mm, Y = 494.3 mm, Z = 498.2 mm,       W = 3.6 deg, P = 7.4 deg,
    GP2:
        UF : 1, UT : 2,
       J1 = 0.0 deg, J2 = 0.0 deg
 };
P[211] {
    GP1:
        UF : 6, UT : 5,     CONFIG: 'N U T, 0, 0, 0',
       X = -442.5 mm, Y = 423.5 mm, Z = 498.2 mm,
       W = 3.6 deg, P = 7.2 deg,
    GP2:
        UF : 1, UT : 2,
       J1 = 0.0 deg, J2 = 0.0 deg
 };
P[483] {
    GP1:
        UF : 6, UT : 5,     CONFIG: 'N U T, 0, 0, 0',
 X = -425.5 mm, Y = 494.5 mm, Z = 498.2 mm,       W = 3.6 deg, P = 7.2 deg,
    GP2:
        UF : 1, UT : 2,
       J1 = 0.0 deg, J2 = 0.0 deg
 };
P[212] {
    GP1:
        UF : 6, UT : 5,     CONFIG: 'N U T, 0, 0, 0',
       X = -442.4 mm, Y = 423.7 mm, Z = 498.2 mm,
       W = 3.8 deg, P = 7.0 deg,
    GP2:
        UF : 1, UT : 2,
       J1 = 0.0 deg, J2 = 0.0 deg
 };
P[484] {
    GP1:
        UF : 6, UT : 5,     CONFIG: 'N U T, 0, 0, 0',
 X = -425.4 mm, Y = 494.7 mm, Z = 498.2 mm,       W = 3.8 deg, P = 7.0 deg,
    GP2:
        UF : 1, UT : 2,
       J1 = 0.0 deg, J2 = 0.0 deg
 };
P[213] {
    GP1:
        UF : 6, UT : 5,     CONFIG: 'N U T, 0, 0, 0',
       X = -441.9 mm, Y = 424.6 mm, Z = 498.2 mm,
       W = 3.6 deg, P = 6.2 deg,
    GP2:
        UF : 1, UT : 2,
       J1 = 0.0 deg, J2 = 0.0 deg
 };
P[485] {
    GP1:
        UF : 6, UT : 5,     CONFIG: 'N U T, 0, 0, 0',
 X = -424.9 mm, Y = 495.6 mm, Z = 498.2 mm,       W = 3.6 deg, P = 6.2 deg,
    GP2:
        UF : 1, UT : 2,
       J1 = 0.0 deg, J2 = 0.0 deg
 };
P[214] {
    GP1:
        UF : 6, UT : 5,     CONFIG: 'N U T, 0, 0, 0',
       X = -441.3 mm, Y = 425.5 mm, Z = 498.2 mm,
       W = 3.7 deg, P = 5.6 deg,
    GP2:
        UF : 1, UT : 2,
       J1 = 0.0 deg, J2 = 0.0 deg
 };
P[486] {
    GP1:
        UF : 6, UT : 5,     CONFIG: 'N U T, 0, 0, 0',
 X = -424.3 mm, Y = 496.5 mm, Z = 498.2 mm,       W = 3.7 deg, P = 5.6 deg,
    GP2:
        UF : 1, UT : 2,
       J1 = 0.0 deg, J2 = 0.0 deg
 };
P[215] {
    GP1:
        UF : 6, UT : 5,     CONFIG: 'N U T, 0, 0, 0',
       X = -441.0 mm, Y = 426.0 mm, Z = 498.2 mm,
       W = 3.6 deg, P = 4.9 deg,
    GP2:
        UF : 1, UT : 2,
       J1 = 0.0 deg, J2 = 0.0 deg
 };
P[487] {
    GP1:
        UF : 6, UT : 5,     CONFIG: 'N U T, 0, 0, 0',
 X = -424.0 mm, Y = 497.0 mm, Z = 498.2 mm,       W = 3.6 deg, P = 4.9 deg,
    GP2:
        UF : 1, UT : 2,
       J1 = 0.0 deg, J2 = 0.0 deg
 };
P[216] {
    GP1:
        UF : 6, UT : 5,     CONFIG: 'N U T, 0, 0, 0',
       X = -440.8 mm, Y = 426.2 mm, Z = 498.2 mm,
       W = 3.5 deg, P = 4.6 deg,
    GP2:
        UF : 1, UT : 2,
       J1 = 0.0 deg, J2 = 0.0 deg
 };
P[488] {
    GP1:
        UF : 6, UT : 5,     CONFIG: 'N U T, 0, 0, 0',
 X = -423.8 mm, Y = 497.2 mm, Z = 498.2 mm,       W = 3.5 deg, P = 4.6 deg,
    GP2:
        UF : 1, UT : 2,
       J1 = 0.0 deg, J2 = 0.0 deg
 };
P[217] {
    GP1:
        UF : 6, UT : 5,     CONFIG: 'N U T, 0, 0, 0',
       X = -440.6 mm, Y = 426.4 mm, Z = 498.2 mm,
       W = 3.4 deg, P = 4.3 deg,
    GP2:
        UF : 1, UT : 2,
       J1 = 0.0 deg, J2 = 0.0 deg
 };
P[489] {
    GP1:
        UF : 6, UT : 5,     CONFIG: 'N U T, 0, 0, 0',
 X = -423.6 mm, Y = 497.4 mm, Z = 498.2 mm,       W = 3.4 deg, P = 4.3 deg,
    GP2:
        UF : 1, UT : 2,
       J1 = 0.0 deg, J2 = 0.0 deg
 };
P[218] {
    GP1:
        UF : 6, UT : 5,     CONFIG: 'N U T, 0, 0, 0',
       X = -439.4 mm, Y = 427.9 mm, Z = 498.2 mm,
       W = 2.8 deg, P = 3.5 deg,
    GP2:
        UF : 1, UT : 2,
       J1 = 0.0 deg, J2 = 0.0 deg
 };
P[490] {
    GP1:
        UF : 6, UT : 5,     CONFIG: 'N U T, 0, 0, 0',
 X = -422.4 mm, Y = 498.9 mm, Z = 498.2 mm,       W = 2.8 deg, P = 3.5 deg,
    GP2:
        UF : 1, UT : 2,
       J1 = 0.0 deg, J2 = 0.0 deg
 };
P[219] {
    GP1:
        UF : 6, UT : 5,     CONFIG: 'N U T, 0, 0, 0',
       X = -432.7 mm, Y = 435.1 mm, Z = 498.2 mm,
       W = 2.7 deg, P = 3.3 deg,
    GP2:
        UF : 1, UT : 2,
       J1 = 0.0 deg, J2 = 0.0 deg
 };
P[491] {
    GP1:
        UF : 6, UT : 5,     CONFIG: 'N U T, 0, 0, 0',
 X = -415.7 mm, Y = 506.1 mm, Z = 498.2 mm,       W = 2.7 deg, P = 3.3 deg,
    GP2:
        UF : 1, UT : 2,
       J1 = 0.0 deg, J2 = 0.0 deg
 };
P[220] {
    GP1:
        UF : 6, UT : 5,     CONFIG: 'N U T, 0, 0, 0',
       X = -425.9 mm, Y = 442.2 mm, Z = 498.2 mm,
       W = 2.5 deg, P = 3.2 deg,
    GP2:
        UF : 1, UT : 2,
       J1 = 0.0 deg, J2 = 0.0 deg
 };
P[492] {
    GP1:
        UF : 6, UT : 5,     CONFIG: 'N U T, 0, 0, 0',
 X = -408.9 mm, Y = 513.2 mm, Z = 498.2 mm,       W = 2.5 deg, P = 3.2 deg,
    GP2:
        UF : 1, UT : 2,
       J1 = 0.0 deg, J2 = 0.0 deg
 };
P[221] {
    GP1:
        UF : 6, UT : 5,     CONFIG: 'N U T, 0, 0, 0',
       X = -419.1 mm, Y = 449.2 mm, Z = 498.2 mm,
       W = 2.4 deg, P = 3.0 deg,
    GP2:
        UF : 1, UT : 2,
       J1 = 0.0 deg, J2 = 0.0 deg
 };
P[493] {
    GP1:
        UF : 6, UT : 5,     CONFIG: 'N U T, 0, 0, 0',
 X = -402.1 mm, Y = 520.2 mm, Z = 498.2 mm,       W = 2.4 deg, P = 3.0 deg,
    GP2:
        UF : 1, UT : 2,
       J1 = 0.0 deg, J2 = 0.0 deg
 };
P[222] {
    GP1:
        UF : 6, UT : 5,     CONFIG: 'N U T, 0, 0, 0',
       X = -412.2 mm, Y = 456.2 mm, Z = 498.2 mm,
       W = 2.3 deg, P = 2.8 deg,
    GP2:
        UF : 1, UT : 2,
       J1 = 0.0 deg, J2 = 0.0 deg
 };
P[494] {
    GP1:
        UF : 6, UT : 5,     CONFIG: 'N U T, 0, 0, 0',
 X = -395.2 mm, Y = 527.2 mm, Z = 498.2 mm,       W = 2.3 deg, P = 2.8 deg,
    GP2:
        UF : 1, UT : 2,
       J1 = 0.0 deg, J2 = 0.0 deg
 };
P[223] {
    GP1:
        UF : 6, UT : 5,     CONFIG: 'N U T, 0, 0, 0',
       X = -405.2 mm, Y = 463.1 mm, Z = 498.2 mm,
       W = 2.1 deg, P = 2.6 deg,
    GP2:
        UF : 1, UT : 2,
       J1 = 0.0 deg, J2 = 0.0 deg
 };
P[495] {
    GP1:
        UF : 6, UT : 5,     CONFIG: 'N U T, 0, 0, 0',
 X = -388.2 mm, Y = 534.1 mm, Z = 498.2 mm,       W = 2.1 deg, P = 2.6 deg,
    GP2:
        UF : 1, UT : 2,
       J1 = 0.0 deg, J2 = 0.0 deg
 };
P[224] {
    GP1:
        UF : 6, UT : 5,     CONFIG: 'N U T, 0, 0, 0',
       X = -398.0 mm, Y = 469.8 mm, Z = 498.2 mm,
       W = 2.0 deg, P = 2.5 deg,
    GP2:
        UF : 1, UT : 2,
       J1 = 0.0 deg, J2 = 0.0 deg
 };
P[496] {
    GP1:
        UF : 6, UT : 5,     CONFIG: 'N U T, 0, 0, 0',
 X = -381.0 mm, Y = 540.8 mm, Z = 498.2 mm,       W = 2.0 deg, P = 2.5 deg,
    GP2:
        UF : 1, UT : 2,
       J1 = 0.0 deg, J2 = 0.0 deg
 };
P[225] {
    GP1:
        UF : 6, UT : 5,     CONFIG: 'N U T, 0, 0, 0',
       X = -390.6 mm, Y = 476.2 mm, Z = 498.2 mm,
       W = 1.8 deg, P = 2.3 deg,
    GP2:
        UF : 1, UT : 2,
       J1 = 0.0 deg, J2 = 0.0 deg
 };
P[497] {
    GP1:
        UF : 6, UT : 5,     CONFIG: 'N U T, 0, 0, 0',
 X = -373.6 mm, Y = 547.2 mm, Z = 498.2 mm,       W = 1.8 deg, P = 2.3 deg,
    GP2:
        UF : 1, UT : 2,
       J1 = 0.0 deg, J2 = 0.0 deg
 };
P[226] {
    GP1:
        UF : 6, UT : 5,     CONFIG: 'N U T, 0, 0, 0',
       X = -386.2 mm, Y = 479.8 mm, Z = 498.2 mm,
       W = 1.8 deg, P = 2.2 deg,
    GP2:
        UF : 1, UT : 2,
       J1 = 0.0 deg, J2 = 0.0 deg
 };
P[498] {
    GP1:
        UF : 6, UT : 5,     CONFIG: 'N U T, 0, 0, 0',
 X = -369.2 mm, Y = 550.8 mm, Z = 498.2 mm,       W = 1.8 deg, P = 2.2 deg,
    GP2:
        UF : 1, UT : 2,
       J1 = 0.0 deg, J2 = 0.0 deg
 };
P[227] {
    GP1:
        UF : 6, UT : 5,     CONFIG: 'N U T, 0, 0, 0',
       X = -384.7 mm, Y = 481.4 mm, Z = 498.2 mm,
       W = 1.7 deg, P = 2.1 deg,
    GP2:
        UF : 1, UT : 2,
       J1 = 0.0 deg, J2 = 0.0 deg
 };
P[499] {
    GP1:
        UF : 6, UT : 5,     CONFIG: 'N U T, 0, 0, 0',
 X = -367.7 mm, Y = 552.4 mm, Z = 498.2 mm,       W = 1.7 deg, P = 2.1 deg,
    GP2:
        UF : 1, UT : 2,
       J1 = 0.0 deg, J2 = 0.0 deg
 };
P[228] {
    GP1:
        UF : 6, UT : 5,     CONFIG: 'N U T, 0, 0, 0',
       X = -383.6 mm, Y = 482.9 mm, Z = 498.2 mm,
       W = 1.7 deg, P = 2.1 deg,
    GP2:
        UF : 1, UT : 2,
       J1 = 0.0 deg, J2 = 0.0 deg
 };
P[500] {
    GP1:
        UF : 6, UT : 5,     CONFIG: 'N U T, 0, 0, 0',
 X = -366.6 mm, Y = 553.9 mm, Z = 498.2 mm,       W = 1.7 deg, P = 2.1 deg,
    GP2:
        UF : 1, UT : 2,
       J1 = 0.0 deg, J2 = 0.0 deg
 };
P[229] {
    GP1:
        UF : 6, UT : 5,     CONFIG: 'N U T, 0, 0, 0',
       X = -383.0 mm, Y = 484.0 mm, Z = 498.2 mm,
       W = 1.7 deg, P = 2.1 deg,
    GP2:
        UF : 1, UT : 2,
       J1 = 0.0 deg, J2 = 0.0 deg
 };
P[501] {
    GP1:
        UF : 6, UT : 5,     CONFIG: 'N U T, 0, 0, 0',
 X = -366.0 mm, Y = 555.0 mm, Z = 498.2 mm,       W = 1.7 deg, P = 2.1 deg,
    GP2:
        UF : 1, UT : 2,
       J1 = 0.0 deg, J2 = 0.0 deg
 };
P[230] {
    GP1:
        UF : 6, UT : 5,     CONFIG: 'N U T, 0, 0, 0',
       X = -382.7 mm, Y = 484.8 mm, Z = 498.2 mm,
       W = 1.7 deg, P = 2.1 deg,
    GP2:
        UF : 1, UT : 2,
       J1 = 0.0 deg, J2 = 0.0 deg
 };
P[502] {
    GP1:
        UF : 6, UT : 5,     CONFIG: 'N U T, 0, 0, 0',
 X = -365.7 mm, Y = 555.8 mm, Z = 498.2 mm,       W = 1.7 deg, P = 2.1 deg,
    GP2:
        UF : 1, UT : 2,
       J1 = 0.0 deg, J2 = 0.0 deg
 };
P[231] {
    GP1:
        UF : 6, UT : 5,     CONFIG: 'N U T, 0, 0, 0',
       X = -382.2 mm, Y = 486.3 mm, Z = 498.2 mm,
       W = 1.7 deg, P = 2.1 deg,
    GP2:
        UF : 1, UT : 2,
       J1 = 0.0 deg, J2 = 0.0 deg
 };
P[503] {
    GP1:
        UF : 6, UT : 5,     CONFIG: 'N U T, 0, 0, 0',
 X = -365.2 mm, Y = 557.3 mm, Z = 498.2 mm,       W = 1.7 deg, P = 2.1 deg,
    GP2:
        UF : 1, UT : 2,
       J1 = 0.0 deg, J2 = 0.0 deg
 };
P[232] {
    GP1:
        UF : 6, UT : 5,     CONFIG: 'N U T, 0, 0, 0',
       X = -382.1 mm, Y = 487.2 mm, Z = 498.2 mm,
       W = 1.7 deg, P = 2.0 deg,
    GP2:
        UF : 1, UT : 2,
       J1 = 0.0 deg, J2 = 0.0 deg
 };
P[504] {
    GP1:
        UF : 6, UT : 5,     CONFIG: 'N U T, 0, 0, 0',
 X = -365.1 mm, Y = 558.2 mm, Z = 498.2 mm,       W = 1.7 deg, P = 2.0 deg,
    GP2:
        UF : 1, UT : 2,
       J1 = 0.0 deg, J2 = 0.0 deg
 };
P[233] {
    GP1:
        UF : 6, UT : 5,     CONFIG: 'N U T, 0, 0, 0',
       X = -382.0 mm, Y = 488.0 mm, Z = 498.2 mm,
       W = 1.6 deg, P = 2.0 deg,
    GP2:
        UF : 1, UT : 2,
       J1 = 0.0 deg, J2 = 0.0 deg
 };
P[505] {
    GP1:
        UF : 6, UT : 5,     CONFIG: 'N U T, 0, 0, 0',
 X = -365.0 mm, Y = 559.0 mm, Z = 498.2 mm,       W = 1.6 deg, P = 2.0 deg,
    GP2:
        UF : 1, UT : 2,
       J1 = 0.0 deg, J2 = 0.0 deg
 };
P[234] {
    GP1:
        UF : 6, UT : 5,     CONFIG: 'N U T, 0, 0, 0',
       X = -382.0 mm, Y = 490.2 mm, Z = 498.2 mm,
       W = 1.6 deg, P = 1.9 deg,
    GP2:
        UF : 1, UT : 2,
       J1 = 0.0 deg, J2 = 0.0 deg
 };
P[506] {
    GP1:
        UF : 6, UT : 5,     CONFIG: 'N U T, 0, 0, 0',
 X = -365.0 mm, Y = 561.2 mm, Z = 498.2 mm,       W = 1.6 deg, P = 1.9 deg,
    GP2:
        UF : 1, UT : 2,
       J1 = 0.0 deg, J2 = 0.0 deg
 };
P[235] {
    GP1:
        UF : 6, UT : 5,     CONFIG: 'N U T, 0, 0, 0',
       X = -382.5 mm, Y = 492.5 mm, Z = 498.2 mm,
       W = 1.5 deg, P = 1.9 deg,
    GP2:
        UF : 1, UT : 2,
       J1 = 0.0 deg, J2 = 0.0 deg
 };
P[507] {
    GP1:
        UF : 6, UT : 5,     CONFIG: 'N U T, 0, 0, 0',
 X = -365.5 mm, Y = 563.5 mm, Z = 498.2 mm,       W = 1.5 deg, P = 1.9 deg,
    GP2:
        UF : 1, UT : 2,
       J1 = 0.0 deg, J2 = 0.0 deg
 };
P[236] {
    GP1:
        UF : 6, UT : 5,     CONFIG: 'N U T, 0, 0, 0',
       X = -383.3 mm, Y = 494.4 mm, Z = 498.2 mm,
       W = 1.5 deg, P = 1.9 deg,
    GP2:
        UF : 1, UT : 2,
       J1 = 0.0 deg, J2 = 0.0 deg
 };
P[508] {
    GP1:
        UF : 6, UT : 5,     CONFIG: 'N U T, 0, 0, 0',
 X = -366.3 mm, Y = 565.4 mm, Z = 498.2 mm,       W = 1.5 deg, P = 1.9 deg,
    GP2:
        UF : 1, UT : 2,
       J1 = 0.0 deg, J2 = 0.0 deg
 };
P[237] {
    GP1:
        UF : 6, UT : 5,     CONFIG: 'N U T, 0, 0, 0',
       X = -384.4 mm, Y = 496.1 mm, Z = 498.2 mm,
       W = 1.5 deg, P = 1.8 deg,
    GP2:
        UF : 1, UT : 2,
       J1 = 0.0 deg, J2 = 0.0 deg
 };
P[509] {
    GP1:
        UF : 6, UT : 5,     CONFIG: 'N U T, 0, 0, 0',
 X = -367.4 mm, Y = 567.1 mm, Z = 498.2 mm,       W = 1.5 deg, P = 1.8 deg,
    GP2:
        UF : 1, UT : 2,
       J1 = 0.0 deg, J2 = 0.0 deg
 };
P[238] {
    GP1:
        UF : 6, UT : 5,     CONFIG: 'N U T, 0, 0, 0',
       X = -386.0 mm, Y = 497.4 mm, Z = 498.2 mm,
       W = 1.5 deg, P = 1.8 deg,
    GP2:
        UF : 1, UT : 2,
       J1 = 0.0 deg, J2 = 0.0 deg
 };
P[510] {
    GP1:
        UF : 6, UT : 5,     CONFIG: 'N U T, 0, 0, 0',
 X = -369.0 mm, Y = 568.4 mm, Z = 498.2 mm,       W = 1.5 deg, P = 1.8 deg,
    GP2:
        UF : 1, UT : 2,
       J1 = 0.0 deg, J2 = 0.0 deg
 };
P[239] {
    GP1:
        UF : 6, UT : 5,     CONFIG: 'N U T, 0, 0, 0',
       X = -388.4 mm, Y = 499.2 mm, Z = 498.2 mm,
       W = 1.4 deg, P = 1.8 deg,
    GP2:
        UF : 1, UT : 2,
       J1 = 0.0 deg, J2 = 0.0 deg
 };
P[511] {
    GP1:
        UF : 6, UT : 5,     CONFIG: 'N U T, 0, 0, 0',
 X = -371.4 mm, Y = 570.2 mm, Z = 498.2 mm,       W = 1.4 deg, P = 1.8 deg,
    GP2:
        UF : 1, UT : 2,
       J1 = 0.0 deg, J2 = 0.0 deg
 };
P[240] {
    GP1:
        UF : 6, UT : 5,     CONFIG: 'N U T, 0, 0, 0',
       X = -396.6 mm, Y = 504.7 mm, Z = 498.2 mm,
       W = 1.3 deg, P = 1.6 deg,
    GP2:
        UF : 1, UT : 2,
       J1 = 0.0 deg, J2 = 0.0 deg
 };
P[512] {
    GP1:
        UF : 6, UT : 5,     CONFIG: 'N U T, 0, 0, 0',
 X = -379.6 mm, Y = 575.7 mm, Z = 498.2 mm,       W = 1.3 deg, P = 1.6 deg,
    GP2:
        UF : 1, UT : 2,
       J1 = 0.0 deg, J2 = 0.0 deg
 };
P[241] {
    GP1:
        UF : 6, UT : 5,     CONFIG: 'N U T, 0, 0, 0',
       X = -404.9 mm, Y = 509.9 mm, Z = 498.2 mm,
       W = 1.1 deg, P = 1.4 deg,
    GP2:
        UF : 1, UT : 2,
       J1 = 0.0 deg, J2 = 0.0 deg
 };
P[513] {
    GP1:
        UF : 6, UT : 5,     CONFIG: 'N U T, 0, 0, 0',
 X = -387.9 mm, Y = 580.9 mm, Z = 498.2 mm,       W = 1.1 deg, P = 1.4 deg,
    GP2:
        UF : 1, UT : 2,
       J1 = 0.0 deg, J2 = 0.0 deg
 };
P[242] {
    GP1:
        UF : 6, UT : 5,     CONFIG: 'N U T, 0, 0, 0',
       X = -413.3 mm, Y = 515.0 mm, Z = 498.2 mm,
       W = 1.0 deg, P = 1.3 deg,
    GP2:
        UF : 1, UT : 2,
       J1 = 0.0 deg, J2 = 0.0 deg
 };
P[514] {
    GP1:
        UF : 6, UT : 5,     CONFIG: 'N U T, 0, 0, 0',
 X = -396.3 mm, Y = 586.0 mm, Z = 498.2 mm,       W = 1.0 deg, P = 1.3 deg,
    GP2:
        UF : 1, UT : 2,
       J1 = 0.0 deg, J2 = 0.0 deg
 };
P[243] {
    GP1:
        UF : 6, UT : 5,     CONFIG: 'N U T, 0, 0, 0',
       X = -421.9 mm, Y = 519.9 mm, Z = 498.2 mm,
       W = 0.9 deg, P = 1.1 deg,
    GP2:
        UF : 1, UT : 2,
       J1 = 0.0 deg, J2 = 0.0 deg
 };
P[515] {
    GP1:
        UF : 6, UT : 5,     CONFIG: 'N U T, 0, 0, 0',
 X = -404.9 mm, Y = 590.9 mm, Z = 498.2 mm,       W = 0.9 deg, P = 1.1 deg,
    GP2:
        UF : 1, UT : 2,
       J1 = 0.0 deg, J2 = 0.0 deg
 };
P[244] {
    GP1:
        UF : 6, UT : 5,     CONFIG: 'N U T, 0, 0, 0',
       X = -430.5 mm, Y = 524.7 mm, Z = 498.2 mm,
       W = 0.7 deg, P = 0.9 deg,
    GP2:
        UF : 1, UT : 2,
       J1 = 0.0 deg, J2 = 0.0 deg
 };
P[516] {
    GP1:
        UF : 6, UT : 5,     CONFIG: 'N U T, 0, 0, 0',
 X = -413.5 mm, Y = 595.7 mm, Z = 498.2 mm,       W = 0.7 deg, P = 0.9 deg,
    GP2:
        UF : 1, UT : 2,
       J1 = 0.0 deg, J2 = 0.0 deg
 };
P[245] {
    GP1:
        UF : 6, UT : 5,     CONFIG: 'N U T, 0, 0, 0',
       X = -439.2 mm, Y = 529.3 mm, Z = 498.2 mm,
       W = 0.6 deg, P = 0.7 deg,
    GP2:
        UF : 1, UT : 2,
       J1 = 0.0 deg, J2 = 0.0 deg
 };
P[517] {
    GP1:
        UF : 6, UT : 5,     CONFIG: 'N U T, 0, 0, 0',
 X = -422.2 mm, Y = 600.3 mm, Z = 498.2 mm,       W = 0.6 deg, P = 0.7 deg,
    GP2:
        UF : 1, UT : 2,
       J1 = 0.0 deg, J2 = 0.0 deg
 };
P[246] {
    GP1:
        UF : 6, UT : 5,     CONFIG: 'N U T, 0, 0, 0',
       X = -441.6 mm, Y = 530.5 mm, Z = 498.2 mm,
       W = 0.6 deg, P = 0.7 deg,
    GP2:
        UF : 1, UT : 2,
       J1 = 0.0 deg, J2 = 0.0 deg
 };
P[518] {
    GP1:
        UF : 6, UT : 5,     CONFIG: 'N U T, 0, 0, 0',
 X = -424.6 mm, Y = 601.5 mm, Z = 498.2 mm,       W = 0.6 deg, P = 0.7 deg,
    GP2:
        UF : 1, UT : 2,
       J1 = 0.0 deg, J2 = 0.0 deg
 };
P[247] {
    GP1:
        UF : 6, UT : 5,     CONFIG: 'N U T, 0, 0, 0',
       X = -443.6 mm, Y = 531.8 mm, Z = 498.2 mm,
       W = 0.5 deg, P = 0.6 deg,
    GP2:
        UF : 1, UT : 2,
       J1 = 0.0 deg, J2 = 0.0 deg
 };
P[519] {
    GP1:
        UF : 6, UT : 5,     CONFIG: 'N U T, 0, 0, 0',
 X = -426.6 mm, Y = 602.8 mm, Z = 498.2 mm,       W = 0.5 deg, P = 0.6 deg,
    GP2:
        UF : 1, UT : 2,
       J1 = 0.0 deg, J2 = 0.0 deg
 };
P[248] {
    GP1:
        UF : 6, UT : 5,     CONFIG: 'N U T, 0, 0, 0',
       X = -445.3 mm, Y = 533.2 mm, Z = 498.2 mm,
       W = 0.5 deg, P = 0.6 deg,
    GP2:
        UF : 1, UT : 2,
       J1 = 0.0 deg, J2 = 0.0 deg
 };
P[520] {
    GP1:
        UF : 6, UT : 5,     CONFIG: 'N U T, 0, 0, 0',
 X = -428.3 mm, Y = 604.2 mm, Z = 498.2 mm,       W = 0.5 deg, P = 0.6 deg,
    GP2:
        UF : 1, UT : 2,
       J1 = 0.0 deg, J2 = 0.0 deg
 };
P[249] {
    GP1:
        UF : 6, UT : 5,     CONFIG: 'N U T, 0, 0, 0',
       X = -446.6 mm, Y = 534.7 mm, Z = 498.2 mm,
       W = 0.5 deg, P = 0.6 deg,
    GP2:
        UF : 1, UT : 2,
       J1 = 0.0 deg, J2 = 0.0 deg
 };
P[521] {
    GP1:
        UF : 6, UT : 5,     CONFIG: 'N U T, 0, 0, 0',
 X = -429.6 mm, Y = 605.7 mm, Z = 498.2 mm,       W = 0.5 deg, P = 0.6 deg,
    GP2:
        UF : 1, UT : 2,
       J1 = 0.0 deg, J2 = 0.0 deg
 };
P[250] {
    GP1:
        UF : 6, UT : 5,     CONFIG: 'N U T, 0, 0, 0',
       X = -448.1 mm, Y = 536.7 mm, Z = 498.2 mm,
       W = 0.4 deg, P = 0.5 deg,
    GP2:
        UF : 1, UT : 2,
       J1 = 0.0 deg, J2 = 0.0 deg
 };
P[522] {
    GP1:
        UF : 6, UT : 5,     CONFIG: 'N U T, 0, 0, 0',
 X = -431.1 mm, Y = 607.7 mm, Z = 498.2 mm,       W = 0.4 deg, P = 0.5 deg,
    GP2:
        UF : 1, UT : 2,
       J1 = 0.0 deg, J2 = 0.0 deg
 };
P[251] {
    GP1:
        UF : 6, UT : 5,     CONFIG: 'N U T, 0, 0, 0',
       X = -453.1 mm, Y = 545.0 mm, Z = 498.2 mm,
       W = 0.3 deg, P = 0.3 deg,
    GP2:
        UF : 1, UT : 2,
       J1 = 0.0 deg, J2 = 0.0 deg
 };
P[523] {
    GP1:
        UF : 6, UT : 5,     CONFIG: 'N U T, 0, 0, 0',
 X = -436.1 mm, Y = 616.0 mm, Z = 498.2 mm,       W = 0.3 deg, P = 0.3 deg,
    GP2:
        UF : 1, UT : 2,
       J1 = 0.0 deg, J2 = 0.0 deg
 };
P[252] {
    GP1:
        UF : 6, UT : 5,     CONFIG: 'N U T, 0, 0, 0',
       X = -454.9 mm, Y = 548.0 mm, Z = 498.2 mm,
       W = 0.2 deg, P = 0.3 deg,
    GP2:
        UF : 1, UT : 2,
       J1 = 0.0 deg, J2 = 0.0 deg
 };
P[524] {
    GP1:
        UF : 6, UT : 5,     CONFIG: 'N U T, 0, 0, 0',
 X = -437.9 mm, Y = 619.0 mm, Z = 498.2 mm,       W = 0.2 deg, P = 0.3 deg,
    GP2:
        UF : 1, UT : 2,
       J1 = 0.0 deg, J2 = 0.0 deg
 };
P[253] {
    GP1:
        UF : 6, UT : 5,     CONFIG: 'N U T, 0, 0, 0',
       X = -456.8 mm, Y = 551.1 mm, Z = 498.2 mm,
       W = 0.2 deg, P = 0.2 deg,
    GP2:
        UF : 1, UT : 2,
       J1 = 0.0 deg, J2 = 0.0 deg
 };
P[525] {
    GP1:
        UF : 6, UT : 5,     CONFIG: 'N U T, 0, 0, 0',
 X = -439.8 mm, Y = 622.1 mm, Z = 498.2 mm,       W = 0.2 deg, P = 0.2 deg,
    GP2:
        UF : 1, UT : 2,
       J1 = 0.0 deg, J2 = 0.0 deg
 };
P[254] {
    GP1:
        UF : 6, UT : 5,     CONFIG: 'N U T, 0, 0, 0',
       X = -457.4 mm, Y = 552.3 mm, Z = 498.2 mm,
       W = 0.2 deg, P = 0.2 deg,
    GP2:
        UF : 1, UT : 2,
       J1 = 0.0 deg, J2 = 0.0 deg
 };
P[526] {
    GP1:
        UF : 6, UT : 5,     CONFIG: 'N U T, 0, 0, 0',
 X = -440.4 mm, Y = 623.3 mm, Z = 498.2 mm,       W = 0.2 deg, P = 0.2 deg,
    GP2:
        UF : 1, UT : 2,
       J1 = 0.0 deg, J2 = 0.0 deg
 };
P[255] {
    GP1:
        UF : 6, UT : 5,     CONFIG: 'N U T, 0, 0, 0',
       X = -457.9 mm, Y = 553.5 mm, Z = 498.2 mm,
       W = 0.2 deg, P = 0.2 deg,
    GP2:
        UF : 1, UT : 2,
       J1 = 0.0 deg, J2 = 0.0 deg
 };
P[527] {
    GP1:
        UF : 6, UT : 5,     CONFIG: 'N U T, 0, 0, 0',
 X = -440.9 mm, Y = 624.5 mm, Z = 498.2 mm,       W = 0.2 deg, P = 0.2 deg,
    GP2:
        UF : 1, UT : 2,
       J1 = 0.0 deg, J2 = 0.0 deg
 };
P[256] {
    GP1:
        UF : 6, UT : 5,     CONFIG: 'N U T, 0, 0, 0',
       X = -458.2 mm, Y = 554.8 mm, Z = 498.2 mm,
       W = 0.1 deg, P = 0.2 deg,
    GP2:
        UF : 1, UT : 2,
       J1 = 0.0 deg, J2 = 0.0 deg
 };
P[528] {
    GP1:
        UF : 6, UT : 5,     CONFIG: 'N U T, 0, 0, 0',
 X = -441.2 mm, Y = 625.8 mm, Z = 498.2 mm,       W = 0.1 deg, P = 0.2 deg,
    GP2:
        UF : 1, UT : 2,
       J1 = 0.0 deg, J2 = 0.0 deg
 };
P[257] {
    GP1:
        UF : 6, UT : 5,     CONFIG: 'N U T, 0, 0, 0',
       X = -458.3 mm, Y = 556.5 mm, Z = 498.2 mm,
       W = 0.1 deg, P = 0.1 deg,
    GP2:
        UF : 1, UT : 2,
       J1 = 0.0 deg, J2 = 0.0 deg
 };
P[529] {
    GP1:
        UF : 6, UT : 5,     CONFIG: 'N U T, 0, 0, 0',
 X = -441.3 mm, Y = 627.5 mm, Z = 498.2 mm,       W = 0.1 deg, P = 0.1 deg,
    GP2:
        UF : 1, UT : 2,
       J1 = 0.0 deg, J2 = 0.0 deg
 };
P[258] {
    GP1:
        UF : 6, UT : 5,     CONFIG: 'N U T, 0, 0, 0',
       X = -458.0 mm, Y = 558.2 mm, Z = 498.2 mm,
       W = 0.1 deg, P = 0.1 deg,
    GP2:
        UF : 1, UT : 2,
       J1 = 0.0 deg, J2 = 0.0 deg
 };
P[530] {
    GP1:
        UF : 6, UT : 5,     CONFIG: 'N U T, 0, 0, 0',
 X = -441.0 mm, Y = 629.2 mm, Z = 498.2 mm,       W = 0.1 deg, P = 0.1 deg,
    GP2:
        UF : 1, UT : 2,
       J1 = 0.0 deg, J2 = 0.0 deg
 };
P[259] {
    GP1:
        UF : 6, UT : 5,     CONFIG: 'N U T, 0, 0, 0',
       X = -457.2 mm, Y = 559.9 mm, Z = 498.2 mm,
       W = 0.1 deg, P = 0.1 deg,
    GP2:
        UF : 1, UT : 2,
       J1 = 0.0 deg, J2 = 0.0 deg
 };
P[531] {
    GP1:
        UF : 6, UT : 5,     CONFIG: 'N U T, 0, 0, 0',
 X = -440.2 mm, Y = 630.9 mm, Z = 498.2 mm,       W = 0.1 deg, P = 0.1 deg,
    GP2:
        UF : 1, UT : 2,
       J1 = 0.0 deg, J2 = 0.0 deg
 };
P[260] {
    GP1:
        UF : 6, UT : 5,     CONFIG: 'N U T, 0, 0, 0',
       X = -456.0 mm, Y = 561.5 mm, Z = 498.2 mm,
       W = 0.0 deg, P = 0.0 deg,
    GP2:
        UF : 1, UT : 2,
       J1 = 0.0 deg, J2 = 0.0 deg
 };
P[532] {
    GP1:
        UF : 6, UT : 5,     CONFIG: 'N U T, 0, 0, 0',
 X = -439.0 mm, Y = 632.5 mm, Z = 498.2 mm,       W = 0.0 deg, P = 0.0 deg,
    GP2:
        UF : 1, UT : 2,
       J1 = 0.0 deg, J2 = 0.0 deg
 };
P[261] {
    GP1:
        UF : 6, UT : 5,     CONFIG: 'N U T, 0, 0, 0',
       X = -454.4 mm, Y = 562.8 mm, Z = 498.2 mm,
       W = 0.0 deg, P = 0.0 deg,
    GP2:
        UF : 1, UT : 2,
       J1 = 0.0 deg, J2 = 0.0 deg
 };
P[533] {
    GP1:
        UF : 6, UT : 5,     CONFIG: 'N U T, 0, 0, 0',
 X = -437.4 mm, Y = 633.8 mm, Z = 498.2 mm,       W = 0.0 deg, P = 0.0 deg,
    GP2:
        UF : 1, UT : 2,
       J1 = 0.0 deg, J2 = 0.0 deg
 };
P[262] {
    GP1:
        UF : 6, UT : 5,     CONFIG: 'N U T, 0, 0, 0',
       X = -446.4 mm, Y = 568.1 mm, Z = 498.2 mm,
       W = 0.0 deg, P = 0.0 deg,
    GP2:
        UF : 1, UT : 2,
       J1 = 0.0 deg, J2 = 0.0 deg
 };
P[534] {
    GP1:
        UF : 6, UT : 5,     CONFIG: 'N U T, 0, 0, 0',
 X = -429.4 mm, Y = 639.1 mm, Z = 498.2 mm,       W = 0.0 deg, P = 0.0 deg,
    GP2:
        UF : 1, UT : 2,
       J1 = 0.0 deg, J2 = 0.0 deg
 };
P[263] {
    GP1:
        UF : 6, UT : 5,     CONFIG: 'N U T, 0, 0, 0',
       X = -438.4 mm, Y = 573.3 mm, Z = 498.2 mm,
       W = 0.0 deg, P = 0.0 deg,
    GP2:
        UF : 1, UT : 2,
       J1 = 0.0 deg, J2 = 0.0 deg
 };
P[535] {
    GP1:
        UF : 6, UT : 5,     CONFIG: 'N U T, 0, 0, 0',
 X = -421.4 mm, Y = 644.3 mm, Z = 498.2 mm,       W = 0.0 deg, P = 0.0 deg,
    GP2:
        UF : 1, UT : 2,
       J1 = 0.0 deg, J2 = 0.0 deg
 };
P[264] {
    GP1:
        UF : 6, UT : 5,     CONFIG: 'N U T, 0, 0, 0',
       X = -430.4 mm, Y = 578.5 mm, Z = 498.2 mm,
       W = 0.0 deg, P = 0.0 deg,
    GP2:
        UF : 1, UT : 2,
       J1 = 0.0 deg, J2 = 0.0 deg
 };
P[536] {
    GP1:
        UF : 6, UT : 5,     CONFIG: 'N U T, 0, 0, 0',
 X = -413.4 mm, Y = 649.5 mm, Z = 498.2 mm,       W = 0.0 deg, P = 0.0 deg,
    GP2:
        UF : 1, UT : 2,
       J1 = 0.0 deg, J2 = 0.0 deg
 };
P[265] {
    GP1:
        UF : 6, UT : 5,     CONFIG: 'N U T, 0, 0, 0',
       X = -422.4 mm, Y = 583.7 mm, Z = 498.2 mm,
       W = 0.0 deg, P = 0.0 deg,
    GP2:
        UF : 1, UT : 2,
       J1 = 0.0 deg, J2 = 0.0 deg
 };
P[537] {
    GP1:
        UF : 6, UT : 5,     CONFIG: 'N U T, 0, 0, 0',
 X = -405.4 mm, Y = 654.7 mm, Z = 498.2 mm,       W = 0.0 deg, P = 0.0 deg,
    GP2:
        UF : 1, UT : 2,
       J1 = 0.0 deg, J2 = 0.0 deg
 };
P[266] {
    GP1:
        UF : 6, UT : 5,     CONFIG: 'N U T, 0, 0, 0',
       X = -414.4 mm, Y = 588.8 mm, Z = 498.2 mm,
       W = 0.0 deg, P = 0.0 deg,
    GP2:
        UF : 1, UT : 2,
       J1 = 0.0 deg, J2 = 0.0 deg
 };
P[538] {
    GP1:
        UF : 6, UT : 5,     CONFIG: 'N U T, 0, 0, 0',
 X = -397.4 mm, Y = 659.8 mm, Z = 498.2 mm,       W = 0.0 deg, P = 0.0 deg,
    GP2:
        UF : 1, UT : 2,
       J1 = 0.0 deg, J2 = 0.0 deg
 };
P[267] {
    GP1:
        UF : 6, UT : 5,     CONFIG: 'N U T, 0, 0, 0',
       X = -406.4 mm, Y = 594.0 mm, Z = 498.2 mm,
       W = 0.0 deg, P = 0.0 deg,
    GP2:
        UF : 1, UT : 2,
       J1 = 0.0 deg, J2 = 0.0 deg
 };
P[539] {
    GP1:
        UF : 6, UT : 5,     CONFIG: 'N U T, 0, 0, 0',
 X = -389.4 mm, Y = 665.0 mm, Z = 498.2 mm,       W = 0.0 deg, P = 0.0 deg,
    GP2:
        UF : 1, UT : 2,
       J1 = 0.0 deg, J2 = 0.0 deg
 };
P[268] {
    GP1:
        UF : 6, UT : 5,     CONFIG: 'N U T, 0, 0, 0',
       X = -398.4 mm, Y = 599.2 mm, Z = 498.2 mm,
       W = 0.0 deg, P = 0.0 deg,
    GP2:
        UF : 1, UT : 2,
       J1 = 0.0 deg, J2 = 0.0 deg
 };
P[540] {
    GP1:
        UF : 6, UT : 5,     CONFIG: 'N U T, 0, 0, 0',
 X = -381.4 mm, Y = 670.2 mm, Z = 498.2 mm,       W = 0.0 deg, P = 0.0 deg,
    GP2:
        UF : 1, UT : 2,
       J1 = 0.0 deg, J2 = 0.0 deg
 };
P[269] {
    GP1:
        UF : 6, UT : 5,     CONFIG: 'N U T, 0, 0, 0',
       X = -390.5 mm, Y = 604.4 mm, Z = 498.2 mm,
       W = 0.0 deg, P = 0.0 deg,
    GP2:
        UF : 1, UT : 2,
       J1 = 0.0 deg, J2 = 0.0 deg
 };
P[541] {
    GP1:
        UF : 6, UT : 5,     CONFIG: 'N U T, 0, 0, 0',
 X = -373.5 mm, Y = 675.4 mm, Z = 498.2 mm,       W = 0.0 deg, P = 0.0 deg,
    GP2:
        UF : 1, UT : 2,
       J1 = 0.0 deg, J2 = 0.0 deg
 };
P[270] {
    GP1:
        UF : 6, UT : 5,     CONFIG: 'N U T, 0, 0, 0',
       X = -382.5 mm, Y = 609.6 mm, Z = 498.2 mm,
       W = 0.0 deg, P = 0.0 deg,
    GP2:
        UF : 1, UT : 2,
       J1 = 0.0 deg, J2 = 0.0 deg
 };
P[542] {
    GP1:
        UF : 6, UT : 5,     CONFIG: 'N U T, 0, 0, 0',
 X = -365.5 mm, Y = 680.6 mm, Z = 498.2 mm,       W = 0.0 deg, P = 0.0 deg,
    GP2:
        UF : 1, UT : 2,
       J1 = 0.0 deg, J2 = 0.0 deg
 };
/END
